{attribute 'GeneratedUsingTerminal: EK1122-0000-0018'}
{attribute addProperty BoxType "EK1122-0000-0018"}
{attribute addProperty Id "RC40_EPP_EPP1322_0001RC40_EPP_EPP1322_0001_ECA1E6F9120"}
{attribute addProperty CRC "3842371207"}
{attribute addProperty Size "120"}
{attribute addProperty Name "RC40_A3 (EK1122)"}
TYPE RC40_A3_EK1122_E505EE87 EXTENDS EK1122_1FC0878B :
STRUCT
	{attribute addProperty Name "RC40_EPP (EPP1322-0001)"}
	{attribute addProperty PreviousPort "RC40_A3 (EK1122) : D"}
	RC40_EPP_EPP1322_0001 : RC40_EPP_EPP1322_0001_ECA1E6F9;
END_STRUCT
END_TYPE

(* stored: Version 1.2.0.0, ProductVersion 3.1.4024.11
   DUT RC40_A3_EK1122_E505EE87: Id {5fd825aa-ba60-00de-0a85-c304d6153216} *)
